//-----------------------------------------------------------------------------------------------------
//																
//									 	Tkmatik sp z o.o.
//
//	Name					:		FB_Save
//	Author					:		AM
//	Release Date			:		12.01.2022
//	Current ver				:		v 0.1
// 	Last correction 		:		12.01.2022
// 
//	Description				:
//		Special FB for saving structures to BINARY files						
//
//	Requared hardware		:
//
// 	Configuration			:
//
//
//-----------------------------------------------------------------------------------------------------

FUNCTION_BLOCK FB_Save
VAR_INPUT
	sFilePath											:	STRING(255);					//	File path (e.g. 'C:\1.txt'
	pStructAdr											:	PVOID;                          //	Pointer on data struct
	udiStructSize										:	UDINT;                          //	Size of datastruct
	bExecute											:	BOOL;                           //
END_VAR                                                                                     
VAR_OUTPUT                                                                                  
	bBusy												:	BOOL;                           //	FB is Busy
	bDone												:	BOOL;                           //	Load cycle done, DATA actual 
	bError												:	BOOL;                           //	Flag error
	nErrId												:	UDINT;                          //	Error ID
END_VAR                                                                                     
VAR                                                                                         
	fbFileOpen											:	FB_FileOpen;                    //	FB for opening 
	fbFileClose											:	FB_FileClose;                   //	FB for closing
	fbFileWrite											:	FB_FileWrite;                   //	FB for saving
	hFile												:	UINT;                           //	File hendler
	eMainCase											:	E_FileOpSteps;                  //	Main cycle case value
	rtExecute											:	R_TRIG;                         //	Rtrig for start
END_VAR

ACT_FBs();
ACT_Main();

ACTION ACT_FBs:
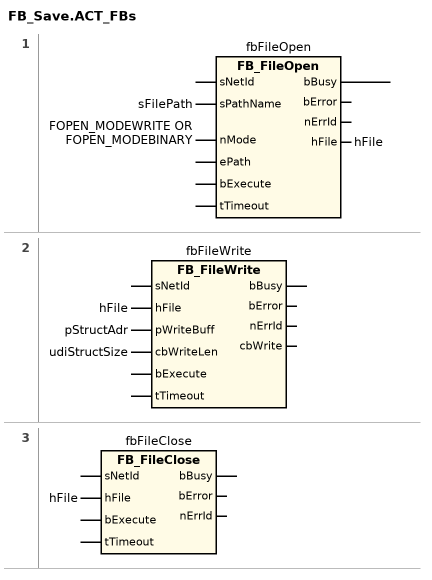
// NETWORK 1
fbFileOpen(sPathName := sFilePath, nMode := FOPEN_MODEWRITE OR FOPEN_MODEBINARY, hFile => hFile); // FB_FileOpen

// NETWORK 2
fbFileWrite(hFile := hFile, pWriteBuff := pStructAdr, cbWriteLen := udiStructSize); // FB_FileWrite

// NETWORK 3
fbFileClose(hFile := hFile); // FB_FileClose
END_ACTION

ACTION ACT_Main:
rtExecute(CLK:=bExecute);
IF (NOT bExecute) THEN
	bDone												:=	FALSE;
END_IF

CASE eMainCase OF
	E_FileOpSteps.eNop:
		fbFileClose.bExecute							:=	FALSE;
		fbFileOpen.bExecute								:=	FALSE;
		fbFileWrite.bExecute							:=	FALSE;
		bBusy											:=	FALSE;
		
		IF (rtExecute.Q) THEN
			bError										:=	FALSE;
			nErrId										:=	0;
			eMainCase									:=	E_FileOpSteps.eStartOpen;
			bBusy										:=	TRUE;
		END_IF
		
	E_FileOpSteps.eStartOpen:
		fbFileOpen.bExecute								:=	TRUE;
		eMainCase										:=	E_FileOpSteps.eWaitOpen;

	E_FileOpSteps.eWaitOpen:
		IF (fbFileOpen.bError) THEN
			bError										:=	TRUE;
			nErrId										:=	10;
			eMainCase									:=	E_FileOpSteps.eNop;
		END_IF
		IF (NOT fbFileOpen.bBusy) THEN
			fbFileOpen.bExecute							:=	FALSE;
			eMainCase									:=	E_FileOpSteps.eStartOper;
		END_IF
		
	E_FileOpSteps.eStartOper:
		fbFileWrite.bExecute							:=	TRUE;
		eMainCase										:=	E_FileOpSteps.eWaitOper;
		
	E_FileOpSteps.eWaitOper:
		IF (fbFileWrite.bError) THEN
			bError										:=	TRUE;
			nErrId										:=	20;
			eMainCase									:=	E_FileOpSteps.eNop;
		END_IF
		IF (NOT fbFileWrite.bBusy) THEN
			fbFileWrite.bExecute						:=	FALSE;
			eMainCase									:=	E_FileOpSteps.eStartClose;
		END_IF
		
	E_FileOpSteps.eStartClose:
		fbFileClose.bExecute							:=	TRUE;
		eMainCase										:=	E_FileOpSteps.eWaitClose;
	
	E_FileOpSteps.eWaitClose:
		IF (fbFileClose.bError) THEN
			bError										:=	TRUE;
			nErrId										:=	30;
			eMainCase									:=	E_FileOpSteps.eNop;
		END_IF
		IF (NOT fbFileClose.bBusy) THEN
			fbFileClose.bExecute						:=	FALSE;
			bDone										:=	TRUE;
			eMainCase									:=	E_FileOpSteps.eNop;
		END_IF	
		
END_CASE
END_ACTION

END_FUNCTION_BLOCK

(* stored: Version 1.1.0.1, ProductVersion 3.1.4026.13, FileIdentifier 6eff2b011f7477dfedc13b0d5fe2b6900b2d0929, FileSignature 6512c3875a6dc0c84b663029aebf3720850ef95e97fea6487409a003f19e0ec04e5cd29122f624442245f7fb6e9f0812f93127b06daa2b30c58adaec163e7eaa5926871741e639ea0e26682353a13ad9c7c402f94fa3d7b41b489cced5cfb34ddbee3c1c2e32671594739f13f6f83b7f000468de9e03d3fafdb1f4eafbb74582f77a2691a33fef9c33edc446d5f044fe71f64f4678a4b322f3656e9c68e1bca5e0707dba4a32281e6a26ec18b2d717f33d5fca4157aa218cdf2804a69360f298c44f929c834bb4f17b2ca5d026a9ddda8434dad2a33c22af24c33e0437179fc6b78ac75d2b7412408a86a260d8c1b6efb8eed3f814914ac397152fc4058a7cc0
   POU FB_Save: Id {d1df88a0-354d-49bf-b591-fed342630838}, SpecialFunc None
   Action ACT_FBs: Id {1d6d8e2b-5ef6-40c5-b346-0734d1f31fd8}
   Action ACT_Main: Id {94a387b3-85bb-45ce-942a-268079ed48d1} *)
